{attribute addProperty BoxType "EL3255-0000-0020"}
{attribute addProperty Id "AI_Compact_Channel_1AT %I*AI_Compact_Channel_2EF51F001620AI_Standard_ChannelAT %I*ARRAY[0..2] OF AI_Standard_Channel_087F71C796120WcStateAT %I*WcState_98A4DF7520.250InfoDataAT %I*InfoData_BC63D37F80100"}
{attribute addProperty CRC "3019552298"}
{attribute addProperty SizeInBites "194"}
{attribute addProperty SizeInBytes "24.25"}
TYPE EL3255_6FD63833 :
STRUCT
	{attribute addProperty Name "AI_Compact_Channel_1"}
	AI_Compact_Channel_1 : AI_Compact_Channel_2EF51F00;
	{attribute addProperty Name "AI_Standard_Channel"}
	AI_Standard_Channel : ARRAY[0..2] OF AI_Standard_Channel_087F71C7;
	{attribute addProperty Name "WcState"}
	WcState : WcState_98A4DF75;
	{attribute addProperty Name "InfoData"}
	InfoData : InfoData_BC63D37F;
END_STRUCT
END_TYPE

(* stored: Version 1.2.0.0, ProductVersion 3.1.4024.9
   DUT EL3255_6FD63833: Id {37186409-4ffd-4cb5-b511-4427fec87fe4} *)
